(* CoDeSys 2.3 export: V2.EXP *)

(* POU V2, ST *)
PROGRAM V2
VAR
	test:INT;
	tmp:BOOL;
	block:EdgeDetection := (onRisingEdge:=1, onFallingEdge:=0);
END_VAR
block(input:=S2_2a, output=>tmp);
IF tmp THEN
	test := test + 1;
END_IF
END_PROGRAM
